(****************************************************************************************)
(*							Beckhoff Automation Poland									*)
(*							L_TBGetBitOfWord v1.0										*)
(*									29.02.2007											*)
(*			This function returns the state of a single bit within a ”word” value		*)
(*______________________________________________________________________________________*)
FUNCTION L_TBGetBitOfWord : BOOL
VAR_INPUT
	wInput:WORD;
	byBitNr:BYTE;
END_VAR
VAR
END_VAR

CASE byBitNr OF
	0:
	L_TBGetBitOfWord:=wInput.0;
	1:
	L_TBGetBitOfWord:=wInput.1;
	2:
	L_TBGetBitOfWord:=wInput.2;
	3:
	L_TBGetBitOfWord:=wInput.3;
	4:
	L_TBGetBitOfWord:=wInput.4;
	5:
	L_TBGetBitOfWord:=wInput.5;
	6:
	L_TBGetBitOfWord:=wInput.6;
	7:
	L_TBGetBitOfWord:=wInput.7;
	8:
	L_TBGetBitOfWord:=wInput.8;
	9:
	L_TBGetBitOfWord:=wInput.9;
	10:
	L_TBGetBitOfWord:=wInput.10;
	11:
	L_TBGetBitOfWord:=wInput.11;
	12:
	L_TBGetBitOfWord:=wInput.12;
	13:
	L_TBGetBitOfWord:=wInput.13;
	14:
	L_TBGetBitOfWord:=wInput.14;
	15:
	L_TBGetBitOfWord:=wInput.15;
END_CASE

END_FUNCTION

(* stored: Version 1.1.0.1, ProductVersion 3.1.4026.13, FileIdentifier a39b4f6258600a423c6bd9da9b053b7607bd0712, FileSignature 9db0c6489ea7e9609fb09c3ba3a487d38c42741eb03f4a26bf1ee4cccd081d8ddd3b997a06d7421ccbd4287ef2463473b010df35feab6da800efa58af3f64b3e47d6d464575d2c471ff8d9ad4cf363487d0b3e5efe7312eab73ae52a449056dc5b7aaf7cb8cd75be75be8abe2bd6a1faf6d2154b976023c380b86f620103b3c6243ef9bbddee97c3f467f8ead6377ec99fa9e6527cf35e6f1093ec5fc4b7e29bddf6cdc638cda5235c2fa39d37307f01ff2aee4cca58b806e5917753cbef3193138718416c2dcf1f272d725acdae7ca299310c99f9f713a12d4f122fca2782fa7b1de6ea4e857e5c289b4fdc4aa2ccad0200fb769ff2743fdb1ac519506fae07
   POU L_TBGetBitOfWord: Id {ade07f71-a1ef-4cec-bcbe-dda4441d0356}, SpecialFunc None *)
